SUBAPPLICATION SubApp_PC_A (* Geraet A (Station 11, 192.168.1.11): 1 SoftKey (Toggle) und GreenWhiteBackground - 'SUB style', das Protokoll steckt im MyLib::sys-Composite (SoftKeyT_PC_A_OPC_Adapter), nicht in der Resource des Geraets - Adapter-Variante von Training_08, gleiche OPC-UA-Adressen wie Training_03 *)
  (* Standard: 61499-2; Description: Copyright (c) 2026 Meisterschulen am Ostbahnhof This program and the accompanying materials are made available under the terms of the Eclipse Public License 2.0 which is available at https://www.eclipse.org/legal/epl-2.0/ SPDX-License-Identifier: EPL-2.0 *)
  (* Version 1.0, 2026-09-04, Franz Höpfinger, Meisterschulen am Ostbahnhof, initial API and implementation and/or initial documentation *)
  PACKAGE subapp::Training_09_OPC_UA_RES;
  IMPORT Uebungen::const::UT::DefaultPool::SoftKey_F1;
  IMPORT VV::const::OPC_UA::myOpcUaAddresses::FF1_TRIGGER_REMOTE_CALL;
  IMPORT VV::const::OPC_UA::myOpcUaAddresses::FF1_STATE_LOCAL_READ;
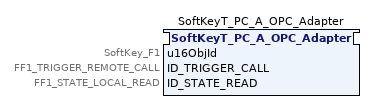
  SUBAPPS
    SoftKeyT_PC_A_OPC_Adapter : MyLib::sys::SoftKeyT_PC_A_OPC_Adapter(u16ObjId := SoftKey_F1, ID_TRIGGER_CALL := FF1_TRIGGER_REMOTE_CALL, ID_STATE_READ := FF1_STATE_LOCAL_READ);
  END_SUBAPPS
END_SUBAPPLICATION
